FUNCTION_BLOCK PID (* PID regulator *)
  (* Version 1.0, AN, SWDC RTSoft *)
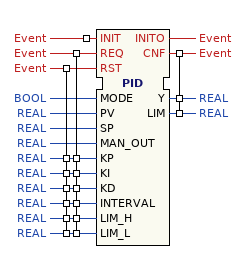
  EVENT_INPUT
    INIT WITH INERROR;
    REQ WITH INERROR, NOISE, KP, KI, KD, INTERVAL, LIM_H, LIM_L;
    RST WITH INERROR, NOISE, KP, KI, KD, INTERVAL, LIM_H, LIM_L;
  END_EVENT
  EVENT_OUTPUT
    INITO;
    CNF WITH Y, LIM;
  END_EVENT
  VAR_INPUT
    MODE : BOOL;
    PV : REAL;
    SP : REAL;
    MAN_OUT : REAL;
    KP : REAL;
    KI : REAL;
    KD : REAL;
    INTERVAL : REAL;
    LIM_H : REAL;
    LIM_L : REAL;
  END_VAR
  VAR_OUTPUT
    Y : REAL;
    LIM : REAL;
  END_VAR
END_FUNCTION_BLOCK
